TYPE "Prod_Part_Area"
VERSION : 0.1
// Block: Prod_Part_Area
   STRUCT
      Halted : Prod_Halted;
      Doors_Closed : Bool;
      Man : Bool;
      CycleON : Bool;
      Running : Bool;
      SetUpDone : Bool;
      SetupDone_Ax : Array[1..14] of Bool;
      MaterialPresenceEntry : Bool;
      MaterialPresenceExit : Bool;
      Material_Presence : Bool;
      MaterialFeedingStandstill : Bool;
      LeadCutMem : Bool;
      Material_Qty_FromLastCut : LReal;
   END_STRUCT;

END_TYPE
